(* Motor Control *)

FUNCTION_BLOCK FB_Motor
  VAR_INPUT
    Start : BOOL;
    Stop : BOOL;
    Reset : BOOL;
    Fault_In : BOOL;
  END_VAR
  VAR_OUTPUT
    Motor_Run : BOOL;
    Motor_Fault : BOOL;
    Motor_Ready : BOOL;
  END_VAR

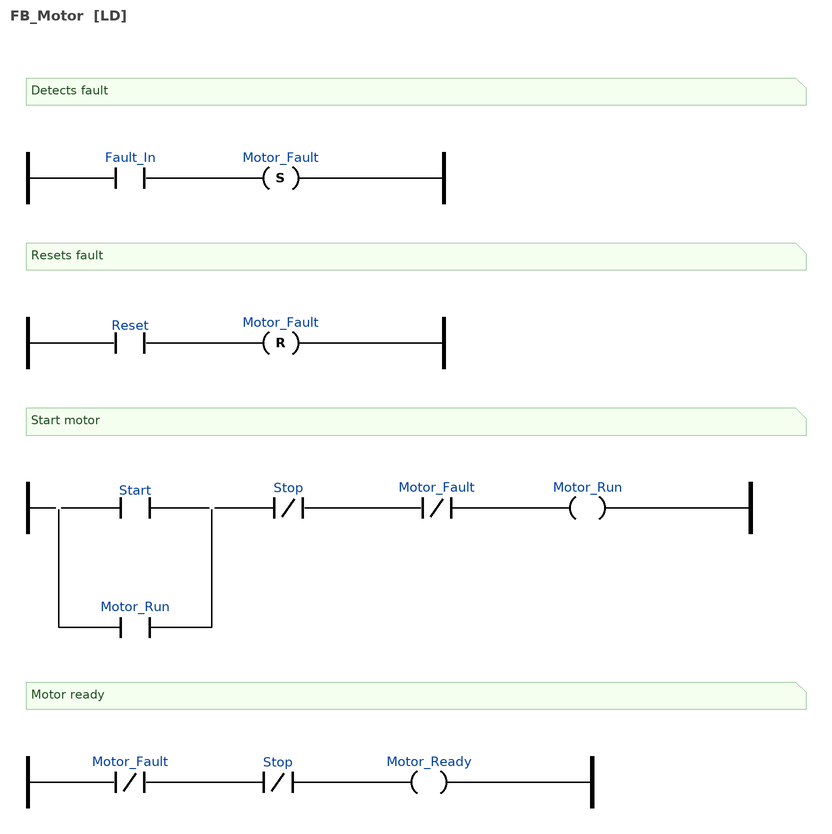
(* LD diagram, written out as Structured Text *)
(* Detects fault *)
IF Fault_In THEN Motor_Fault := TRUE; END_IF;
(* Resets fault *)
IF Reset THEN Motor_Fault := FALSE; END_IF;
(* Start motor *)
Motor_Run := (Start OR Motor_Run) AND NOT Stop AND NOT Motor_Fault;
(* Motor ready *)
Motor_Ready := NOT Motor_Fault AND NOT Stop;
END_FUNCTION_BLOCK
